TYPE ST_ProcessingData :
STRUCT
    // 列
    lrColFirstRowPosition : LREAL;
    lrColGapOfEachRow : LREAL;
    // 行
    lrEvenRowStartPosition : LREAL;
    lrEvenRowInVeloPosition : LREAL;
    lrEvenRowTakePhotoPosition : LREAL;
    lrEvenRowStopPhotoPosition : LREAL;
    lrEvenRowEndConstantSpdPosition : LREAL;
    lrEvenRowStopMovePosition : LREAL;
    // 行
    lrOddRowStartPosition : LREAL;
    lrOddRowInVeloPosition : LREAL;
    lrOddRowTakePhotoPosition : LREAL;
    lrOddRowStopPhotoPosition : LREAL;
    lrOddRowEndConstantSpdPosition : LREAL;
    lrOddRowStopMovePosition : LREAL;
    // 流程
    udiTotalRows : UDINT;
    udiCurrentRow : UDINT;
    udiRemainingRows : UDINT;
    lrCompletePercentage : LREAL;
    bBusy,
    bError,
    bDone,
    bPaused : BOOL;
END_STRUCT
END_TYPE

(* stored: Version 1.1.0.1, ProductVersion 3.1.4024.12
   DUT ST_ProcessingData: Id {b5c9963d-6f9d-4526-a19b-374e5030d44b} *)
